FUNCTION_BLOCK FB_DualMotor IMPLEMENTS I_Motor

VAR
	fMotorSpeed : REAL := 1000;
	bRunning : BOOL;
END_VAR

METHOD Start : BOOL
VAR_INPUT
END_VAR
Start := bRunning := TRUE;
END_METHOD

METHOD Stop : BOOL
VAR_INPUT
END_VAR
Stop := bRunning := FALSE;
END_METHOD

END_FUNCTION_BLOCK

(* stored: Version 1.1.0.1, ProductVersion 3.1.4024.16
   POU FB_DualMotor: Id {52033dc5-5929-42fa-ba5c-1f1619f8ed6f}, SpecialFunc None
   Method Start: Id {135d20c2-00f8-4454-aed8-d14427e6c927}
   Method Stop: Id {d75f9ca8-8fe5-46cf-9497-2414014ce950} *)
